// TIA Portal V16 export
// export: Created 2022-11-14T17:35:41.1379193Z, ExportSetting WithDefaults, DisplayName Totally Integrated Automation Portal, DisplayVersion V16, DisplayName TIA Portal Version Control Interface, DisplayVersion V16, DisplayName TIA Portal Openness, DisplayVersion V16, DisplayName STEP 7 Professional, DisplayVersion V16, DisplayName STEP 7 Safety, DisplayVersion V16, DisplayName WinCC Advanced, DisplayVersion V16
DATA_BLOCK "DB10_ExtConveyors"   // DB10
{ S7_Optimized_Access := 'FALSE' }
VERSION : 0.1
// stored: AutoNumber false, IsOnlyStoredInLoadMemory false, IsWriteProtectedInAS false
   VAR RETAIN
      V1000_0 : Bool := FALSE;
      V1000_1 : Bool := FALSE;
      V1000_2 : Bool := FALSE;
      V1000_3 : Bool := FALSE;
      V1000_4 : Bool := FALSE;
      V1000_5 : Bool := FALSE;
      V1000_6 : Bool := FALSE;
      V1000_7 : Bool := FALSE;
      V1001_0 : Bool := FALSE;
      V1001_1 : Bool := FALSE;
      V1001_2 : Bool := FALSE;
      V1001_3 : Bool := FALSE;
      V1001_4 : Bool := FALSE;
      V1001_5 : Bool := FALSE;
      V1001_6 : Bool := FALSE;
      V1001_7 : Bool := FALSE;
      Out_ConvPos1 : Bool := FALSE;   // Conveyor pos1 motor
      Out_ConvPos2 : Bool := FALSE;   // Conveyor pos2 motor
      Out_ConvPos3 : Bool := FALSE;   // Conveyor pos3 motor
      Out_ConvPos4 : Bool := FALSE;   // Conveyor pos4 motor
      Out_ConvPos5 : Bool := FALSE;   // Conveyor pos5 motor
      Out_ConvPos6 : Bool := FALSE;   // Conveyor pos6 motor
      Out_ConvPos7 : Bool := FALSE;   // Conveyor pos7 motor
      Out_ConvPos8 : Bool := FALSE;   // Conveyor pos8 motor
      Out_ConvPos1Rev : Bool := FALSE;   // Conveyor pos1 motor reverse
      Out_ConvPos2Rev : Bool := FALSE;   // Conveyor pos2 motor reverse
      Out_ConvPos3Rev : Bool := FALSE;   // Conveyor pos3 motor reverse
      Out_ConvPos4Rev : Bool := FALSE;   // Conveyor pos4 motor reverse
      V1003_4 : Bool := FALSE;
      V1003_5 : Bool := FALSE;
      V1003_6 : Bool := FALSE;
      V1003_7 : Bool := FALSE;
      VW1004 : Int := 0;
      Out_ConvPos1X2 : Bool := FALSE;   // Conveyor pos1 motor speed selection X2
      Out_ConvPos2X2 : Bool := FALSE;   // Conveyor pos2 motor speed selection X2
      Out_ConvPos3X2 : Bool := FALSE;   // Conveyor pos3 motor speed selection X2
      Out_ConvPos4X2 : Bool := FALSE;   // Conveyor pos4 motor speed selection X2
      V1006_4 : Bool := FALSE;
      V1006_5 : Bool := FALSE;
      V1006_6 : Bool := FALSE;
      V1006_7 : Bool := FALSE;
      Out_ConvPos2Upw : Bool := FALSE;   // Conveyor pos2 motor upward
      Out_ConvPos2Downw : Bool := FALSE;   // Conveyor pos2 downstroke valve command
      In_ConvPos2Up : Bool := TRUE;   // Conveyor pos2 up photocell NC
      In_ConvPos2Down : Bool := TRUE;   // Conveyor pos2 down photocell NC
      In_ConvPos2ExUp : Bool := TRUE;   // Conveyor pos2 up extrastroke switch NC
      In_ConvPos2Safety : Bool := TRUE;   // Conveyor pos2 down foot safety switch NC
      V1007_6 : Bool := FALSE;
      V1007_7 : Bool := FALSE;
   END_VAR
BEGIN
END_DATA_BLOCK
